{attribute 'qualified_only'}
VAR_GLOBAL PERSISTENT
	pMainJibCylinder : ST_pValveControlledCylinder;				//Parameters for MainJibCylinder uses values from ST_pValveControlledCylinder
	pKnuckleJibCylinder : ST_pValveControlledCylinder; 			//Parameters for KnuckleJib uses values from ST_pValveControlledCylinderv
	pKingRotationCylinder : ST_pValveControlledCylinder;        //Parameters for KingRotation uses values from ST_pValveControlledCylinderv
END_VAR

(* stored: Version 1.1.0.1, ProductVersion 3.1.4024.9
   GVL Param: Id {8cc71902-54f3-4068-b684-2ff92871ee93} *)
